{attribute 'qualified_only'}
{attribute 'strict'}
TYPE ENUM_DiagPaddle :
(
	UNKNOWN := 0,
	PARK :=1,
	UP := 2,
	CENTER := 3,
	PINHOLE := 4,
	DIODE := 5,
	YAG1 := 6,
	YAG2 := 7,
	YAG3 := 8,
	KNIFE := 9
);
END_TYPE

(* stored: Version 1.1.0.1, ProductVersion 3.1.4024.6
   DUT ENUM_DiagPaddle: Id {4b57537f-d152-4dff-a52e-35a4f00e9e55} *)
